FUNCTION_BLOCK SafetyEmergencyStopsWidget
VAR_INPUT
END_VAR
VAR_OUTPUT
	actualStatus : StatusWidget;
END_VAR
VAR_IN_OUT
	ref : SafetyEmergencyStops;
END_VAR
VAR
END_VAR


actualStatus(text  := ref.actualStatus,
             color := HealthBusyToColor(healthStatus := ref.statuses.healthStatus, busyStatus := ref.statuses.busyStatus));

END_FUNCTION_BLOCK

(* stored: Version 1.1.0.1, ProductVersion 3.1.4018.5
   POU SafetyEmergencyStopsWidget: Id {f4ff4b53-922d-4176-b74d-4a73e677f524}, SpecialFunc None *)
